FUNCTION_BLOCK MECH1_DIAG (* Diagnostic for a Unidirectional Mechanism (Clocked) *)
  (* Standard: 61499-1; Classification: Diagnostics; ApplicationDomain: Mechanisms *)
  (* Version 0.1, 2004-10-20, JHC, Rockwell Automation, Renamed to replace old MECH1_DIAG. *)
  (* Version 0.0, 2004-09-26, JHC, Rockwell Automation, Derived from MECH2_DIAG; made composite, incorporated clock. *)
  (* Compiler header: package fb.rt.mva; import fb.rt.math.*; *)
  (* Compiler Java Sun JDK 1.4.2 *)
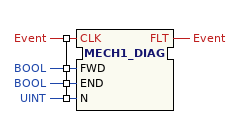
  EVENT_INPUT
    CLK WITH END, FWD, N; (* Diagnostic Clock *)
  END_EVENT
  EVENT_OUTPUT
    FLT; (* Fault Indication *)
  END_EVENT
  VAR_INPUT
    FWD : BOOL; (* Forward Actuation Command from Controller *)
    END : BOOL; (* END(Fully Advanced)Sensor *)
    N : UINT; (* Timeout Period in CLK cycles *)
  END_VAR
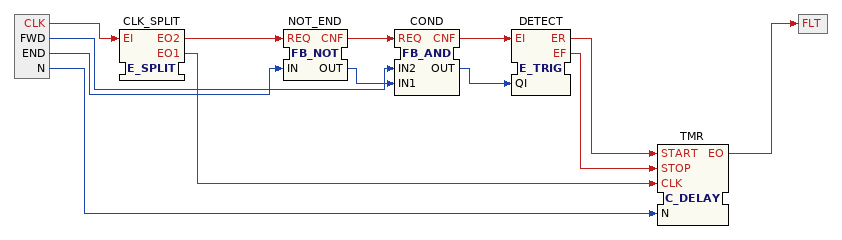
  FBS
    TMR : C_DELAY;
    DETECT : E_TRIG;
    COND : FB_AND;
    NOT_END : FB_NOT;
    CLK_SPLIT : E_SPLIT;
  END_FBS
  EVENT_CONNECTIONS
    DETECT.ER TO TMR.START;
    DETECT.EF TO TMR.STOP;
    COND.CNF TO DETECT.EI;
    NOT_END.CNF TO COND.REQ;
    TMR.EO TO FLT;
    CLK TO CLK_SPLIT.EI;
    CLK_SPLIT.EO2 TO NOT_END.REQ;
    CLK_SPLIT.EO1 TO TMR.CLK;
  END_CONNECTIONS
  DATA_CONNECTIONS
    COND.OUT TO DETECT.QI;
    FWD TO COND.IN2;
    NOT_END.OUT TO COND.IN1;
    END TO NOT_END.IN;
    N TO TMR.N;
  END_CONNECTIONS
END_FUNCTION_BLOCK
